{attribute 'qualified_only'}
VAR_GLOBAL
	//Module C1A2
	ioControl : ioBundleControl;
	ioSafety : ioBundleSafety;

	cylinderControls : ARRAY[1..11] OF RunCylinder;
	signalControls : ARRAY[1..13] OF RunSignal;
	axisControls: ARRAY[1..13] OF RunAxis;
	//
	materialSlots : ARRAY[1..4] OF RunMaterial;	//C1,A1,A2,A3
	stations : ARRAY[1..9] OF POINTER TO RunUnitGeneric;
		
	interfaceControl : InterfaceControlV1;
	InterfaceManual : InterfaceManualV1;
	
	bObjectsLinked : BOOL;
END_VAR

(* stored: Version 1.1.0.1, ProductVersion 3.1.4022.10
   GVL GVL: Id {e607aa11-c301-416f-9cbc-bc4f43af5299} *)
